FUNCTION_BLOCK T_AddMoreThanSizeOfCollectionFalse EXTENDS T_UnitTestBase
VAR
  list : T_ComponentsCollection(3);
  newComponent : ARRAY [1..5] OF T_ComponentMock;
  expected, actual : UDINT;
  result, resultAddOutOfBoundary : BOOL;
END_VAR

list.AddComponent(newComponent[1]);
list.AddComponent(newComponent[2]);
list.AddComponent(newComponent[3]);

resultAddOutOfBoundary := NOT list.AddComponent(newComponent[4]);

expected := 3;
actual := list.Count;

assertion.AssertEquals_UDINT(expected, actual, 'actual := list.Count');
assertion.AssertEquals_BOOL(TRUE, resultAddOutOfBoundary, 'resultAddOutOfBoundary');
TestFinished();

END_FUNCTION_BLOCK

(* stored: Version 1.1.0.1, ProductVersion 3.1.4024.12
   POU T_AddMoreThanSizeOfCollectionFalse: Id {593c008c-f0f7-4432-bc82-f9a0098d8bbc}, SpecialFunc None *)
